Staubli VAL3: trackErr_init.pgx

program trackErr_init()
  local num l_nI
begin
  // This program initialize all variables
  //
  // Input parameters
  //  None            :
  //
  // Output parameters
  //  None            :
  //
  //----------------------------------------------------------------
  //
  // Booleans
  _bSentToHome=false
  _bMutexCnvQueue[0]=false
  _bIsPicking=false
  _bIsPlacing=false
  //

  //
  // Numerical
  _nID[0]=-1
  _nCntBypassed[0]=nBypass[0]


  _nPushIndexTQ[0]=0
  _nPullIndexTQ[0]=0
  _nTimer=0

  for _nCycleTimeIndx=0 to 9
    _nCycleTime[_nCycleTimeIndx]=0
  endFor
  _nCycleTimeIndx=0
  //
  // Points
  pPick.trsf={0,0,0,0,0,0}

  //
  // Transfer Queues
  for l_nI=0 to size(_oTransferQueue,2)-1
    _oTransferQueue[0,l_nI].nID=-1
    _oTransferQueue[0,l_nI].trTrsf={0,0,0,0,0,0}
    _oTransferQueue[0,l_nI].nLatchedValue=0
  endFor
  //
  // Strings
  _sCycleStatus=""
end
